{attribute 'linkalways'} 
{attribute 'no_explicit_call' := 'This FB is a CLASS and must be accessed using methods or properties'}
{attribute 'enable_dynamic_creation'}
FUNCTION_BLOCK ABSTRACT UserDefinedDatatypeBase EXTENDS DatatypeBase IMPLEMENTS I_UserDefinedDatatype
VAR
END_VAR

PROPERTY PUBLIC ABSTRACT Identifier : T_MAXSTRING
GET
END_GET
END_PROPERTY

PROPERTY PUBLIC IsUserDefined : BOOL
GET
IsUserDefined := TRUE;
END_GET
END_PROPERTY

METHOD PROTECTED OnSerializeTypeWith
VAR_INPUT
	Serializer : I_Serializer;
END_VAR
SUPER^.OnSerializeTypeWith(Serializer);
Serializer.AddKeyString('identifier',Identifier);
END_METHOD

METHOD PUBLIC TryCopyFrom : BOOL
VAR_INPUT
	Source : I_Datatype;
END_VAR
VAR
	sourceAsUdt : I_UserDefinedDatatype;
END_VAR
IF NOT __QUERYINTERFACE(Source, sourceAsUdt) THEN
	RETURN;
END_IF

IF sourceAsUdt.Identifier <> Identifier THEN
	RETURN;
END_IF

TryCopyFrom := SUPER^.TryCopyFrom(Source);
END_METHOD

END_FUNCTION_BLOCK

(* stored: Version 1.1.0.1, ProductVersion 3.1.4024.12
   POU UserDefinedDatatypeBase: Id {55e04311-6046-0326-1b5b-d143bc2974cf}, SpecialFunc None
   Folder Protected: Id {2a921985-b010-00e4-0f7a-b7642debd7b7}
   Property Identifier: Id {502a5f15-d89b-0f8d-0c65-99b984a67087}
   Get Get: Id {7bd248e0-f12f-0361-07d7-f79c13979fc4}
   Property IsUserDefined: Id {164d1cf2-f703-4acc-9484-666a26254dab}
   Get Get: Id {c50956ad-91da-48d1-86bd-9c0a6d4a100d}
   Method OnSerializeTypeWith: Id {476ebd9b-4cc5-0045-27b8-a42929a121d4}
   Method TryCopyFrom: Id {04470212-2e7a-4fdf-9649-5ed37bb2ce21} *)
